(* Logix 5000 project; controller BORE Emulate 5570 rev 33.11; software revision 33.00 *)

TASK MainTask (continuous, watchdog 500 ms) : MainProgram, Model

MODULES
   Local : Emulate 5570 (ICP 2, rev 33.11)
       : 1756-IB16 (ICP 3, rev 3.1, Input RPI 20 ms)
       : vendor 1 type 7 code 16 (ICP 4, rev 3.1, Output RPI 20 ms)
END_MODULES

VAR_GLOBAL   (* controller tags *)
   ENGAGE_CLAMP_SW : ALIAS FOR Local:3:I.Data.1;
   LS_CLAMP1_ENGAGED : ALIAS FOR Local:3:I.Data.11;
   LS_CLAMP2_ENGAGED : ALIAS FOR Local:3:I.Data.12;
   LS_DOWN : ALIAS FOR Local:3:I.Data.2;
   LS_UP : ALIAS FOR Local:3:I.Data.3;
   PART_PE : ALIAS FOR Local:3:I.Data.0;
   SAFETY_GATE : ALIAS FOR Local:3:I.Data.10;
   SOL_CLAMP1 : ALIAS FOR Local:4:O.Data.10;
   SOL_CLAMP2 : ALIAS FOR Local:4:O.Data.11;
   SOL_DOWN : ALIAS FOR Local:4:O.Data.1;
   SOL_UP : ALIAS FOR Local:4:O.Data.2;
   SPINDLE_ON : ALIAS FOR Local:4:O.Data.0;
   START_SIGNAL : ALIAS FOR Local:3:I.Data.14;
END_VAR

PROGRAM MainProgram   (* main routine MainRoutine *)
VAR
   CYCLE_COMPLETE_CR : BOOL;   // CYCLE COMPLETED CONTROL RELAY
   CYCLE_IN_PROGRESS_CR : BOOL;   // CYCLE IN PROGRESS CONTROL RELAY
   CYCLE_START_CR : BOOL;
   DOWN_CR : BOOL;   // DOWN CONTROL RELAY
   UP_CR : BOOL;   // UP CONTROL RELAY
END_VAR

ROUTINE MainRoutine   (* ladder *)
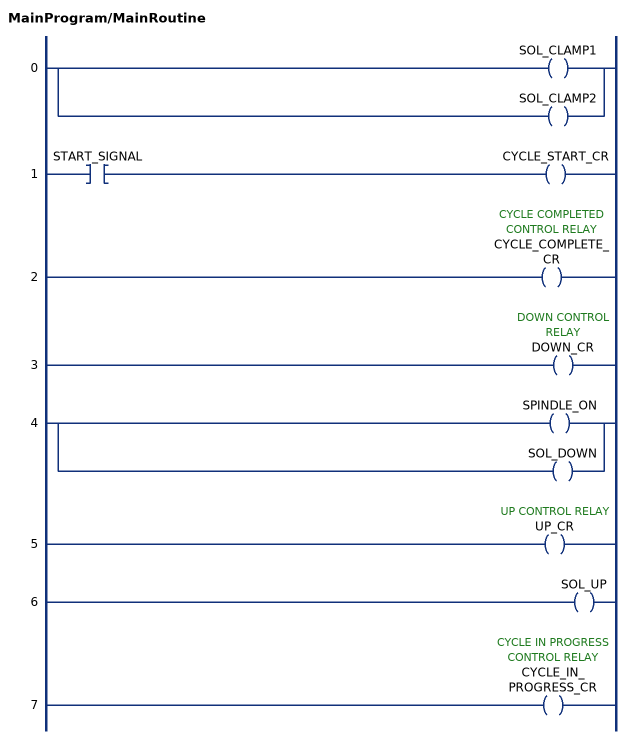
   0: [OTE(SOL_CLAMP1) ,OTE(SOL_CLAMP2) ];
   1: XIC(START_SIGNAL)OTE(CYCLE_START_CR);
   2: OTE(CYCLE_COMPLETE_CR);
   3: OTE(DOWN_CR);
   4: [OTE(SPINDLE_ON) ,OTE(SOL_DOWN) ];
   5: OTE(UP_CR);
   6: OTE(SOL_UP);
   7: OTE(CYCLE_IN_PROGRESS_CR);
END_ROUTINE
END_PROGRAM

PROGRAM Model   (* main routine Emulation *)
VAR
   Clamp1_Sol_Dwell : TIMER := (PRE := 2250);
   Clamp2_Sol_Dwell : TIMER := (PRE := 1500);
   Down_Linit_SW_Dwell : TIMER := (PRE := 1000);
   Down_Travel_Dwell : TIMER := (PRE := 10000);
   Spindle_Carriage : DINT;
   Spindle_Position : DINT;
   Up_Travel_Dwell : TIMER := (PRE := 10000);
END_VAR

ROUTINE Emulation   (* ladder *)
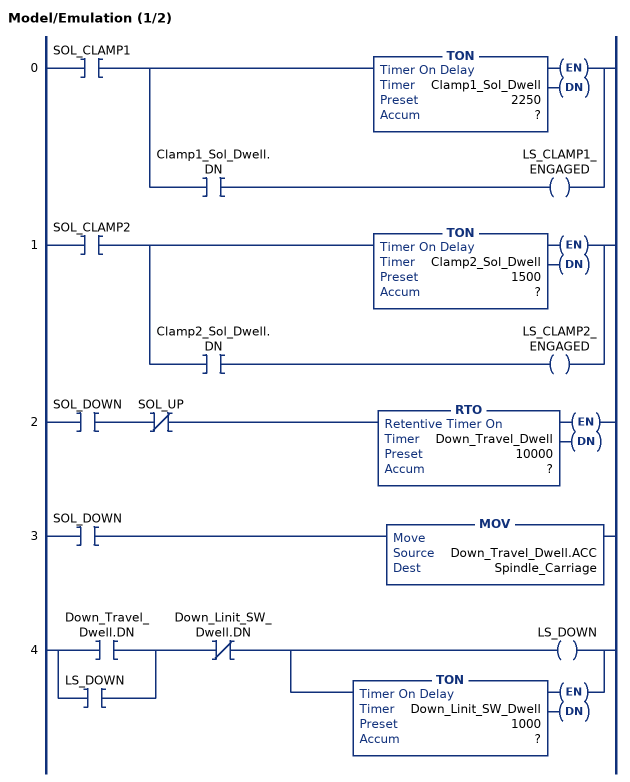
   0: XIC(SOL_CLAMP1)[TON(Clamp1_Sol_Dwell,?,?) ,XIC(Clamp1_Sol_Dwell.DN) OTE(LS_CLAMP1_ENGAGED) ];
   1: XIC(SOL_CLAMP2)[TON(Clamp2_Sol_Dwell,?,?) ,XIC(Clamp2_Sol_Dwell.DN) OTE(LS_CLAMP2_ENGAGED) ];
   2: XIC(SOL_DOWN)XIO(SOL_UP)RTO(Down_Travel_Dwell,?,?);
   3: XIC(SOL_DOWN)MOV(Down_Travel_Dwell.ACC,Spindle_Carriage);
   4: [XIC(Down_Travel_Dwell.DN) ,XIC(LS_DOWN) ]XIO(Down_Linit_SW_Dwell.DN)[OTE(LS_DOWN) ,TON(Down_Linit_SW_Dwell,?,?) ];
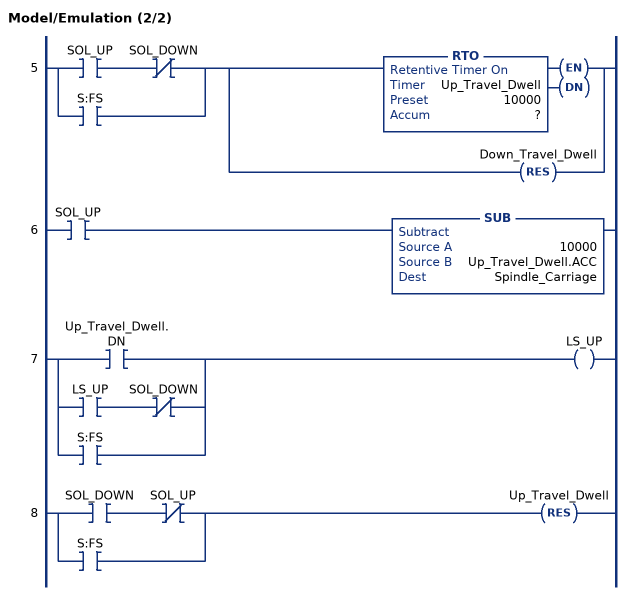
   5: [XIC(SOL_UP) XIO(SOL_DOWN) ,XIC(S:FS) ][RTO(Up_Travel_Dwell,?,?) ,RES(Down_Travel_Dwell) ];
   6: XIC(SOL_UP)SUB(10000,Up_Travel_Dwell.ACC,Spindle_Carriage);
   7: [XIC(Up_Travel_Dwell.DN) ,XIC(LS_UP) XIO(SOL_DOWN) ,XIC(S:FS) ]OTE(LS_UP);
   8: [XIC(SOL_DOWN) XIO(SOL_UP) ,XIC(S:FS) ]RES(Up_Travel_Dwell);
END_ROUTINE
END_PROGRAM
